SUBAPPLICATION Uebung_002a3_AX (* DigitalInput_I1/_I2 mit OR auf DigitalOutput_Q1, mit Plug and Socket *)
  (* Standard: 61499-2; Description: Copyright (c) 2023 Meisterschulen am Ostbahnhof This program and the accompanying materials are made available under the terms of the Eclipse Public License 2.0 which is available at https://www.eclipse.org/legal/epl-2.0/ SPDX-License-Identifier: EPL-2.0 *)
  (* Version 1.0, 2023-10-23, Franz Höpfinger, Meisterschulen am Ostbahnhof *)
  IMPORT logiBUS::io::DI::logiBUS_DI;
  IMPORT logiBUS::io::DI::logiBUS_DI_Events;
  IMPORT logiBUS::io::DQ::logiBUS_DO;
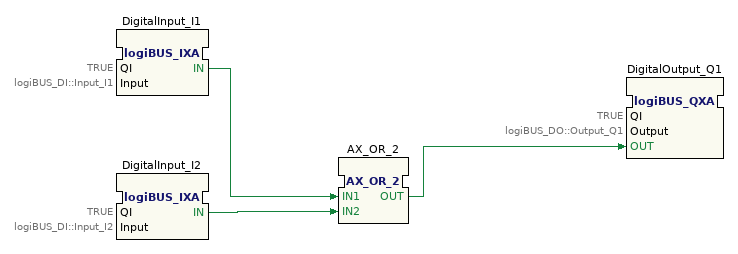
  FBS
    DigitalInput_I1 : logiBUS::io::DI::logiBUS_IXA(QI := TRUE, Input := logiBUS_DI::Input_I1);
    DigitalOutput_Q1 : logiBUS::io::DQ::logiBUS_QXA(QI := TRUE, Output := logiBUS_DO::Output_Q1);
    AX_OR_2 : AX_OR_2;
    DigitalInput_I2 : logiBUS::io::DI::logiBUS_IXA(QI := TRUE, Input := logiBUS_DI::Input_I2);
  END_FBS
  ADAPTER_CONNECTIONS
    AX_OR_2.OUT TO DigitalOutput_Q1.OUT;
    DigitalInput_I1.IN TO AX_OR_2.IN1;
    DigitalInput_I2.IN TO AX_OR_2.IN2;
  END_CONNECTIONS
END_SUBAPPLICATION
